KUKA KRL program: DAI_BEFORE_ZERO_DEVI.src, DAI_BEFORE_ZERO_DEVI.dat

--- DAI_BEFORE_ZERO_DEVI.src ---
&ACCESS RVP
&REL 25
&COMMENT dai_robot_check
&PARAM DISKPATH = KRC:\R1\H_Prog
DEF DAI_BEFORE_ZERO_DEVI( )
;FOLD INI;%{PE}
  ;FOLD BASISTECH INI
    GLOBAL INTERRUPT DECL 3 WHEN $STOPMESS==TRUE DO IR_STOPM ( )
    INTERRUPT ON 3
    BAS (#INITMOV,0 )
  ;ENDFOLD (BASISTECH INI)
  ;FOLD USER INI
    ;Make your modifications here
  ;ENDFOLD (USER INI)
;ENDFOLD (INI)
;FOLD ; Anlagenbezeichn: HC51_B    Stations-Nr: 040RB_100;%{PE}
;FOLD Parameters ;%{h}
;Params IlfProvider=kukaroboter.basistech.inlineforms.comments.comment; Kuka.Content=Anlagenbezeichn: HC51_B    Stations-Nr: 040RB_100
;ENDFOLD
;ENDFOLD
;FOLD ; Stand / Version: V1.0;%{PE}
;FOLD Parameters ;%{h}
;Params IlfProvider=kukaroboter.basistech.inlineforms.comments.comment; Kuka.Content=Stand / Version: V1.0
;ENDFOLD
;ENDFOLD
;FOLD ; Name Bearbeiter: EBZ-AE;%{PE}
;FOLD Parameters ;%{h}
;Params IlfProvider=kukaroboter.basistech.inlineforms.comments.comment; Kuka.Content=Name Bearbeiter: EBZ-AE
;ENDFOLD
;ENDFOLD
;FOLD ; Translator Version:29.01.2024 - Version 15.08;%{PE}
;FOLD Parameters ;%{h}
;Params IlfProvider=kukaroboter.basistech.inlineforms.comments.comment; Kuka.Content=Translator Version:29.01.2024 - Version 15.08
;ENDFOLD
;ENDFOLD

REPEAT
;fold MSG_T1
MSG_SHOW("DAI_H_Prog",#quit,999,"dai_rob_ok_0")
;endfold
; ***************************************
; A C H T U N G !!! Nur in $T1 abfahren
; ***************************************
UNTIL $T1 == TRUE

;FOLD PTP HOME Vel=100 % DEFAULT;%{PE}
;FOLD Parameters ;%{h}
;Params IlfProvider=kukaroboter.basistech.inlineforms.movement.old; Kuka.IsGlobalPoint=False; Kuka.PointName=HOME; Kuka.BlendingEnabled=False; Kuka.MoveDataPtpName=DEFAULT; Kuka.VelocityPtp=100; Kuka.CurrentCDSetIndex=0; Kuka.MovementParameterFieldEnabled=True; IlfCommand=PTP
;ENDFOLD
$BWDSTART = FALSE
PDAT_ACT = PDEFAULT
FDAT_ACT = FHOME
BAS(#PTP_PARAMS, 100.0)
SET_CD_PARAMS (0)
PTP XHOME
;ENDFOLD

WHILE TRUE
 ;fold Satzanwahl / block selection
MSG_BTN("OK")
MSG_SHOW("DAI_H_Prog",#dialog,1,"dai_before_zero_1",handle,answer)
;endfold
; **************************************************
; zum Anfahren der Nullstellung Satzzeiger setzen
HALT
; **************************************************
ENDWHILE

; Kerben anfahren
;FOLD MSG_BTN
MSG_BTN("OK")
MSG_SHOW("DAI_H_Prog",#dialog,3,"dai_before_zero_3",handle,answer)
;ENDFOLD

;FOLD PTP VORJUS_A1 Vel=100 % DEFAULT Tool[64]:Zero Base[64]:Zero ;%{PE}
;FOLD Parameters ;%{h}
;Params IlfProvider=kukaroboter.basistech.inlineforms.movement.old; Kuka.IsGlobalPoint=False; Kuka.PointName=VORJUS_A1; Kuka.BlendingEnabled=False; Kuka.MoveDataPtpName=DEFAULT; Kuka.VelocityPtp=100; Kuka.CurrentCDSetIndex=0; Kuka.MovementParameterFieldEnabled=True; IlfCommand=PTP
;ENDFOLD
$BWDSTART = FALSE
PDAT_ACT = PDEFAULT
FDAT_ACT = FVORJUS_A1
BAS(#PTP_PARAMS, 100.0)
SET_CD_PARAMS (0)
PTP XVORJUS_A1
;ENDFOLD

; Justage Achse 1
halt

;FOLD ; ------------------------------;%{PE}%R 3.2.24,%MKUKATPBASIS,%CCOMMENT,%VNORMAL,%P 2:------------------------------
;ENDFOLD
;FOLD ; Nullstellung Achse 1 mit Werkzeug ;%{PE}
;FOLD Parameters ;%{h}
;Params IlfProvider=kukaroboter.basistech.inlineforms.comments.comment; Kuka.Content=Nullstellung Achse 1 mit Werkzeug
;ENDFOLD
;ENDFOLD

; Kerben anfahren
;FOLD MSG_BTN
MSG_BTN("OK")
MSG_SHOW("DAI_H_Prog",#dialog,3,"dai_before_zero_3",handle,answer)
;ENDFOLD

;FOLD PTP VORJUS Vel=100 % DEFAULT Tool[64]:Zero Base[64]:Zero ;%{PE}
;FOLD Parameters ;%{h}
;Params IlfProvider=kukaroboter.basistech.inlineforms.movement.old; Kuka.IsGlobalPoint=False; Kuka.PointName=VORJUS; Kuka.BlendingEnabled=False; Kuka.MoveDataPtpName=DEFAULT; Kuka.VelocityPtp=100; Kuka.CurrentCDSetIndex=0; Kuka.MovementParameterFieldEnabled=True; IlfCommand=PTP
;ENDFOLD
$BWDSTART = FALSE
PDAT_ACT = PDEFAULT
FDAT_ACT = FVORJUS
BAS(#PTP_PARAMS, 100.0)
SET_CD_PARAMS (0)
PTP XVORJUS
;ENDFOLD

; Justage Achse 2-6
halt

WHILE TRUE
 ;fold Satzanwahl / block selection
MSG_BTN("OK")
MSG_SHOW("DAI_H_Prog",#dialog,1,"dai_before_zero_1",handle,answer)
;endfold
; **************************************************
; zum Anfahren der Nullstellung Achse 2-6 Satzzeiger setzen
HALT
; **************************************************
ENDWHILE

;FOLD ; ------------------------------ ;%{PE}
;FOLD Parameters ;%{h}
;Params IlfProvider=kukaroboter.basistech.inlineforms.comments.comment; Kuka.Content=------------------------------
;ENDFOLD
;ENDFOLD
;FOLD ; Nullstellung Achse 2-6 mit Werkzeug ;%{PE}
;FOLD Parameters ;%{h}
;Params IlfProvider=kukaroboter.basistech.inlineforms.comments.comment; Kuka.Content=Nullstellung Achse 2-6 mit Werkzeug
;ENDFOLD
;ENDFOLD

;FOLD PTP HP010 Vel=100 % PDAT6 Tool[64]:Zero Base[64]:Zero ;%{PE}
;FOLD Parameters ;%{h}
;Params IlfProvider=kukaroboter.basistech.inlineforms.movement.old; Kuka.IsGlobalPoint=False; Kuka.PointName=HP010; Kuka.BlendingEnabled=False; Kuka.MoveDataPtpName=PDAT6; Kuka.VelocityPtp=100; Kuka.CurrentCDSetIndex=0; Kuka.MovementParameterFieldEnabled=True; IlfCommand=PTP
;ENDFOLD
$BWDSTART = FALSE
PDAT_ACT = PPDAT6
FDAT_ACT = FHP010
BAS(#PTP_PARAMS, 100.0)
SET_CD_PARAMS (0)
PTP XHP010
;ENDFOLD

;FOLD PTP HOME Vel=100 % DEFAULT;%{PE}
;FOLD Parameters ;%{h}
;Params IlfProvider=kukaroboter.basistech.inlineforms.movement.old; Kuka.IsGlobalPoint=False; Kuka.PointName=HOME; Kuka.BlendingEnabled=False; Kuka.MoveDataPtpName=DEFAULT; Kuka.VelocityPtp=100; Kuka.CurrentCDSetIndex=0; Kuka.MovementParameterFieldEnabled=True; IlfCommand=PTP
;ENDFOLD
$BWDSTART = FALSE
PDAT_ACT = PDEFAULT
FDAT_ACT = FHOME
BAS(#PTP_PARAMS, 100.0)
SET_CD_PARAMS (0)
PTP XHOME
;ENDFOLD

 ;Collision detection - Off
 ;FOLD COLLDETECT Off ;%{PE}
 ;FOLD Parameters ;%{h}
 ;Params IlfProvider=kukaroboter.basistech.inlineforms.colldetect.off; CollDetect.Command=Off
 ;ENDFOLD
 USE_CD_PARAMS(0)
 ;ENDFOLD

END

--- DAI_BEFORE_ZERO_DEVI.dat ---
&ACCESS RVO
&REL 13
&COMMENT dai_robot_check
&PARAM DISKPATH = KRC:\R1\H_Prog
DEFDAT  DAI_BEFORE_ZERO_DEVI
;FOLD EXTERNAL DECLARATIONS;%{PE}%MKUKATPBASIS,%CEXT,%VCOMMON,%P
;FOLD BASISTECH EXT;%{PE}%MKUKATPBASIS,%CEXT,%VEXT,%P
EXT  BAS (BAS_COMMAND  :IN,REAL  :IN )
DECL INT SUCCESS
;ENDFOLD (BASISTECH EXT)
;FOLD USER EXT;%{E}%MKUKATPUSER,%CEXT,%VEXT,%P
;Make your modifications here
;ENDFOLD (USER EXT)
;FOLD COLLISION
EXT  COLLSTOP (INT  :IN,INT  :IN )
;ENDFOLD  (Collision)
;ENDFOLD (EXTERNAL DECLERATIONS)
DECL INT handle,answer
;//-- Default Dai_ILF Structure SpotWeld --
DECL DSG_Simple_para_T DSG_Simple_para_TDefault={GunNo 1,EQ_Para 3} ;// iW6
;//-- Default Dai_ILF Structure SpotWeld --

; BASIS_SUGG_T declarations
DECL BASIS_SUGG_T LAST_BASIS={POINT1[] "P0                      ",POINT2[] "P0                      ",CP_PARAMS[] "CPDAT0                  ",PTP_PARAMS[] "PDAT0                   ",CONT[] "                        ",CP_VEL[] "2.0                     ",PTP_VEL[] "100                     ",SYNC_PARAMS[] "SYNCDAT                 ",SPL_NAME[] "S0                      ",A_PARAMS[] "ADAT0                   "}

DECL E6AXIS XVORJUS={A1 0.0,A2 -99.0000,A3 101.000,A4 2.50000,A5 2.50000,A6 2.50000,E1 -250.000,E2 0.0,E3 0.0,E4 0.0,E5 0.0,E6 0.0}
DECL E6AXIS XVORJUS_A1={A1 -24.0000,A2 -120.000,A3 55.0000,A4 15.0000,A5 100.000,A6 95.0000,E1 -250.000,E2 0.0,E3 0.0,E4 0.0,E5 0.0,E6 0.0}

; E6POS declarations
DECL E6POS XHP010={X 1302.40588,Y -7.11551,Z 2433.60620,A -95.7493210,B 12.5095587,C -108.084335,S 18,T 2,E1 -250.000,E2 0.0,E3 0.0,E4 0.0,E5 0.0,E6 0.0}
; FDAT declarations
DECL FDAT FHOME={TOOL_NO 64,BASE_NO 64,IPO_FRAME #BASE,POINT2[] " "}
DECL FDAT FVORJUS_A1={TOOL_NO 64,BASE_NO 64,IPO_FRAME #BASE,POINT2[] " "}
DECL FDAT FHP010={TOOL_NO 64,BASE_NO 64,IPO_FRAME #BASE,POINT2[] " "}
DECL FDAT FVORJUS={TOOL_NO 64,BASE_NO 64,IPO_FRAME #BASE,POINT2[] " "}
; MODULEPARAM_T declarations
DECL MODULEPARAM_T LAST_TP_PARAMS={PARAMS[] "Kuka.VelocityPtp=100; Kuka.BlendingEnabled=False; Kuka.CurrentCDSetIndex=0; Dai.IlfConfig=DaiWeldIlfConfig.xml; Dai.IlfTech=DSG_Weld; Kuka.PointName=VORJUS_A1; Kuka.FrameData.base_no=64; Kuka.FrameData.tool_no=64; Kuka.FrameData.ipo_frame=#BASE; Kuka.FrameData.point2=; Kuka.isglobalpoint=False; Kuka.MoveDataPtpName=PDAT6; Kuka.MovementDataPdat.apo_mode=#CDIS; Kuka.MovementDataPdat.apo_dist=0; Kuka.MovementData.vel=100; Kuka.MovementData.acc=100; Kuka.MovementData.gear_jerk=100; Kuka.MovementData.exax_ign=0; Kuka.APXEnabled=False; Kuka.Content=------------------------------     "}
; PDAT declarations
DECL PDAT PPDAT6={VEL 100.000,ACC 100.000,APO_DIST 0.0,APO_MODE #CDIS,GEAR_JERK 50.0000,EXAX_IGN 0}

ENDDAT
